// TIA Portal V19 export
TYPE "LEXCHANGETRAY_typeScanner_sim"
// stored: Access Published
   STRUCT
      simActive : Bool;
      simNG : Bool;
   END_STRUCT;
END_TYPE
